{attribute addProperty BoxType "EL1254--0000"}
{attribute addProperty Id "Status3AT %I*USINT81172Status4AT %I*USINT81173Status1AT %I*USINT81174Status2AT %I*USINT81175LatchPos1AT %I*ULINT648176LatchNeg1AT %I*ULINT648184LatchPos2AT %I*ULINT648192LatchNeg2AT %I*ULINT648200LatchPos3AT %I*ULINT648208LatchNeg3AT %I*ULINT648216LatchPos4AT %I*ULINT648224LatchNeg4AT %I*ULINT648232"}
{attribute addProperty CRC "3189947159"}
{attribute addProperty SizeInBites "544"}
{attribute addProperty SizeInBytes "68"}
TYPE Latch_BE22BB17 :
STRUCT
	{attribute addProperty Name "Status3"}
	Status3 AT %I* : USINT;
	{attribute addProperty Name "Status4"}
	Status4 AT %I* : USINT;
	{attribute addProperty Name "Status1"}
	Status1 AT %I* : USINT;
	{attribute addProperty Name "Status2"}
	Status2 AT %I* : USINT;
	{attribute addProperty Name "LatchPos1"}
	LatchPos1 AT %I* : ULINT;
	{attribute addProperty Name "LatchNeg1"}
	LatchNeg1 AT %I* : ULINT;
	{attribute addProperty Name "LatchPos2"}
	LatchPos2 AT %I* : ULINT;
	{attribute addProperty Name "LatchNeg2"}
	LatchNeg2 AT %I* : ULINT;
	{attribute addProperty Name "LatchPos3"}
	LatchPos3 AT %I* : ULINT;
	{attribute addProperty Name "LatchNeg3"}
	LatchNeg3 AT %I* : ULINT;
	{attribute addProperty Name "LatchPos4"}
	LatchPos4 AT %I* : ULINT;
	{attribute addProperty Name "LatchNeg4"}
	LatchNeg4 AT %I* : ULINT;
END_STRUCT
END_TYPE

(* stored: Version 1.2.0.0, ProductVersion 3.1.4024.9
   DUT Latch_BE22BB17: Id {5fd7b893-e573-4138-928d-91756d548544} *)
